(* Logix 5000 project; controller Timers_TON_TOF_RTO Emulate 5570 rev 30.12; software revision 30.01 *)

TASK MainTask (continuous, watchdog 500 ms) : MainProgram

MODULES
   Local : Emulate 5570 (ICP 2, rev 30.12)
END_MODULES

PROGRAM MainProgram   (* main routine MainRoutine *)
VAR
   Motor1 : BOOL;
   Motor2 : BOOL;
   Motor3 : BOOL;
   Motor4 : BOOL;
   Motor5 : BOOL;
   Motor6 : BOOL;
   PB1 : BOOL;
   PB2 : BOOL;
   PB3 : BOOL;
   PB4 : BOOL;
   PB5 : BOOL;
   PB6 : BOOL;
   Timer1 : TIMER := (PRE := 20000);
   Timer2 : TIMER := (PRE := 10000);
   Timer3 : TIMER := (PRE := 5000);
   Timer4 : TIMER := (PRE := 10000);
   Timer5 : TIMER := (PRE := 10000);
END_VAR

ROUTINE MainRoutine   (* ladder *)
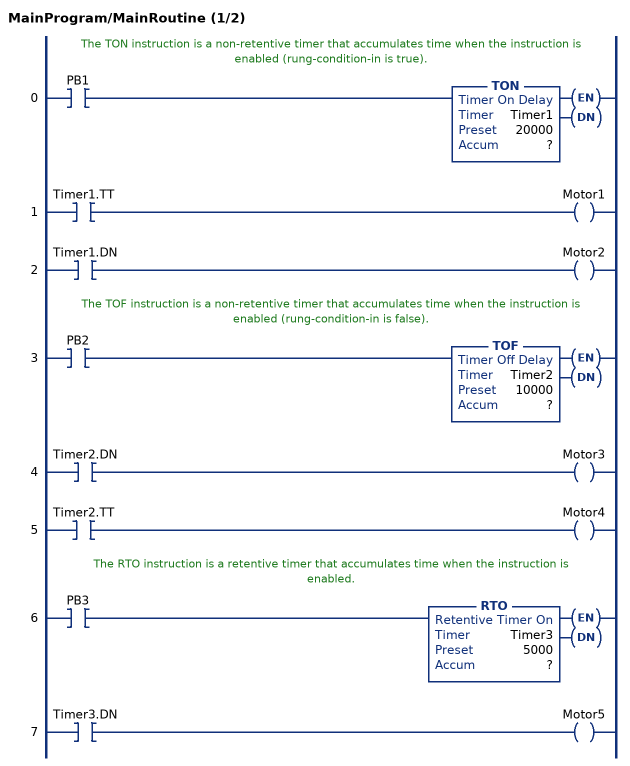
   // The TON instruction is a non-retentive timer that accumulates time when the instruction is enabled (rung-condition-in is true).
   0: XIC(PB1)TON(Timer1,?,?);
   1: XIC(Timer1.TT)OTE(Motor1);
   2: XIC(Timer1.DN)OTE(Motor2);
   // The TOF instruction is a non-retentive timer that accumulates time when the instruction is enabled (rung-condition-in is false).
   3: XIC(PB2)TOF(Timer2,?,?);
   4: XIC(Timer2.DN)OTE(Motor3);
   5: XIC(Timer2.TT)OTE(Motor4);
   // The RTO instruction is a retentive timer that accumulates time when the instruction is enabled.
   6: XIC(PB3)RTO(Timer3,?,?);
   7: XIC(Timer3.DN)OTE(Motor5);
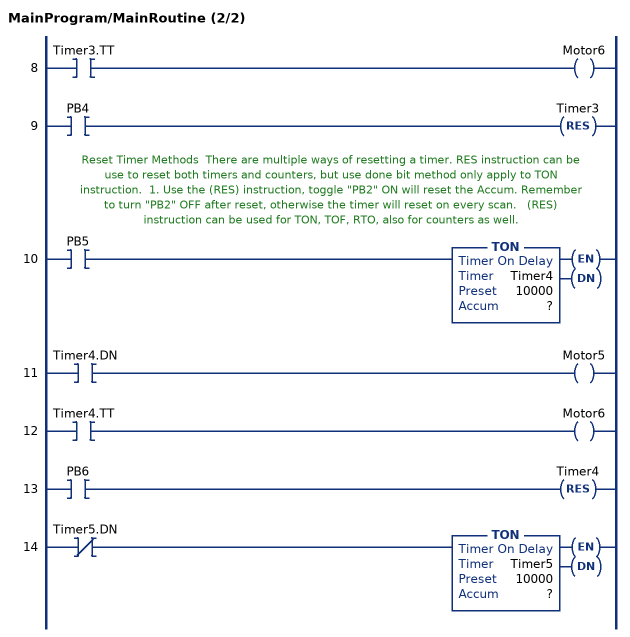
   8: XIC(Timer3.TT)OTE(Motor6);
   9: XIC(PB4)RES(Timer3);
   // Reset Timer Methods  There are multiple ways of resetting a timer. RES instruction can be use to reset both timers and counters, but use done bit method only apply to TON instruction.  1. Use the (RES) instruction, toggle "PB2" ON will reset the Accum. Remember to turn "PB2" OFF after reset, otherwise the timer will reset on every scan.   (RES) instruction can be used for TON, TOF, RTO, also for counters as well.
   10: XIC(PB5)TON(Timer4,?,?);
   11: XIC(Timer4.DN)OTE(Motor5);
   12: XIC(Timer4.TT)OTE(Motor6);
   13: XIC(PB6)RES(Timer4);
   14: XIO(Timer5.DN)TON(Timer5,?,?);
END_ROUTINE
END_PROGRAM
